TYPE HMI_ERR_TemplateClean :
STRUCT
	(*
		Rules:
		Errors shall only be off type BOOL
		Errors shall be set >> the HMI block will do the resetting

		Syntax convention:
		a clear variable name which describes the error			as described below
		InitNotEmpty:BOOL;										//Error [machinepart]: not empty during initialisation
		
		prio's: emergency stop items == 100, e-circuit=99, default (nothing specified) = 50
		adjust as needed
		//example how to pre-set error priorities for the HMI. Default errors get prio 50, Recommend prio 100 for e-stop buttons etc
		ExampleErrorPreConfiggedPrio:BOOL;					//Error[prio=90] Example error with preconfigured prio (key only used at first creation/adding to the HMI-alarm-list-file)
	*)
END_STRUCT
END_TYPE

(* stored: Version 1.1.0.1
   DUT HMI_ERR_TemplateClean: Id {1fccee74-822e-45e1-802f-d0869fc47113} *)
